Yaskawa INFORM job: R1_W27-A3(90,0)OK-KM.JBI

/JOB
//NAME R1_W27-A3(90,0)OK-KM
///FOLDERNAME KRIS-SCIANA
//POS
///NPOS 43,43,0,3,0,0
///TOOL 0
///POSTYPE PULSE
///PULSE
C00000=4830,83199,5771,6899,94988,75055
C00001=-9773,79383,9827,16212,95277,69552
C00002=-9773,79383,9827,16212,95277,-53372
C00003=-9773,-28468,-43390,16212,95277,-53372
C00004=-118130,28395,29263,-77612,79106,-42908
C00005=-118130,42832,63459,-80282,76069,-36632
C00006=-121022,40509,60957,-80752,74157,-36980
C00007=-122076,40550,60998,-80949,73435,-37043
C00008=-122717,40599,61051,-81070,72994,-37080
C00009=-122076,40550,60998,-80949,73435,-37043
C00010=-122043,47472,68552,-81246,73253,-36526
C00011=-122055,44833,65640,-81126,73325,-36733
C00012=-121022,40509,60957,-80752,74157,-36980
C00013=-118130,28395,29263,-77612,79106,-42908
C00014=-120301,29173,30032,-77655,77552,-43056
C00015=-120039,32113,44650,-90901,76713,-36723
C00016=-120861,32104,44640,-91018,76127,-36728
C00017=-119313,33187,45743,-90820,77231,-36662
C00018=-119853,35892,48525,-90967,76837,-36513
C00019=-119313,33187,45743,-90820,77231,-36662
C00020=-118868,30790,31644,-84323,85642,-41471
C00021=-130429,-11916,41219,-108053,40291,-28638
C00022=-116428,-13316,-7274,-52109,62616,-45524
C00023=-117742,-2204,1538,-51719,62054,-45954
C00024=-115860,2997,30006,-91299,52035,-28528
C00025=-121469,1006,3731,-50735,60158,-46989
C00026=-120227,302,2593,-50891,61069,-46816
C00027=-115745,-1819,28231,-92358,52111,-27726
C00028=-112555,-4087,35757,-96933,59618,-24349
C00029=-112542,-4035,35819,-96942,59654,-24342
C00030=-111238,-10662,2688,-62879,64047,-42529
C00031=-111998,-8144,-211,-53563,64102,-43814
C00032=-114545,-38172,-18809,-58928,38901,31311
C00033=-120615,-32838,-15388,-55575,35611,29062
C00034=-102867,26964,48378,-82054,78500,40282
C00035=-119784,-31977,-14810,-55883,36152,29279
C00036=-120619,-32587,-15219,-55544,35624,29044
C00037=-102846,27333,48386,-82014,78545,40201
C00038=-102203,45516,96371,-91697,68609,49479
C00039=-95028,10215,48172,-86436,71799,45925
C00040=-80780,-67431,-36414,-60607,42164,32637
C00041=-21077,34801,-6145,-35147,72854,61023
C00042=19629,104504,14492,-17788,93778,80377
BC00000=161822,1138,1029509
BC00001=179661,1053,1007237
BC00002=277355,1053,807792
BC00003=277355,1053,807792
BC00004=398174,15,734423
BC00005=398174,15,734423
BC00006=398174,15,734423
BC00007=398174,15,734423
BC00008=398174,15,734423
BC00009=398174,15,734423
BC00010=398174,15,734423
BC00011=398174,15,734423
BC00012=398174,15,734423
BC00013=398174,15,734423
BC00014=398174,15,718477
BC00015=396635,15,712098
BC00016=396635,15,712098
BC00017=396635,15,712098
BC00018=396635,15,712098
BC00019=396635,15,712098
BC00020=398174,10910,727845
BC00021=398174,19843,1075175
BC00022=363223,15,893026
BC00023=359892,15,870362
BC00024=358663,16,873958
BC00025=358560,15,861296
BC00026=358560,15,861296
BC00027=358663,16,873958
BC00028=358610,15,874107
BC00029=358610,15,874108
BC00030=358643,15,874329
BC00031=363273,15,905837
BC00032=348983,15,797430
BC00033=344731,15,795268
BC00034=343031,15,794403
BC00035=343031,15,794403
BC00036=343031,15,794403
BC00037=343031,15,644273
BC00038=343031,15,794403
BC00039=343387,15,790284
BC00040=348817,15,727589
BC00041=229605,324,912929
BC00042=148325,534,1039296
///POSTYPE BASE
///RECTAN
///RCONF 0,0,0,0,1,0,0,0,0,0,0,0,0,0,0,0,0,0,0,0,0,0,0,0
P00006=2.006,1.622,-0.565,0.0000,0.0000,0.0000
///RCONF 0,0,0,0,0,0,0,0,0,0,0,0,0,0,0,0,0,0,0,0,0,0,0,0
P00025=3.643,0.007,-2.585,0.0000,0.0000,0.0000
P00026=2.644,0.055,-2.583,0.0000,0.0000,0.0000
//INST
///DATE 2025/04/11 12:42
///ATTR SC,RW
///GROUP1 RB1,BS1
NOP
SFTOF
MOVJ C00000 BC00000 VJ=100.00
MOVJ C00001 BC00001 VJ=100.00
MOVJ C00002 BC00002 VJ=100.00
MOVJ C00003 BC00003 VJ=100.00
MOVL C00004 BC00004 V=1000.0
MOVL C00005 BC00005 V=1000.0
MOVL C00006 BC00006 V=250.0
MOVL C00007 BC00007 V=100.0
REFP 3 C00008 BC00008
CALL JOB:SEARCH-R1
SET P026 P006
SFTON P026
MOVL C00009 BC00009 V=60.0
REFP 3 C00010 BC00010
CALL JOB:SEARCH-R1
SET P026 P006
SFTON P026
MOVL C00011 BC00011 V=60.0
MOVL C00012 BC00012 V=166.7
SFTOF
MOVL C00013 BC00013 V=1000.0
MOVL C00014 BC00014 V=250.0
MOVL C00015 BC00015 V=100.0
REFP 3 C00016 BC00016
CALL JOB:SEARCH-R1
SET P025 P006
SFTON P025
MOVL C00017 BC00017 V=60.0
REFP 3 C00018 BC00018
CALL JOB:SEARCH-R1
SET P025 P006
SFTON P025
MOVL C00019 BC00019 V=60.0
MOVL C00020 BC00020 V=166.7
'Path VIA1038
SFTOF
MOVL C00021 BC00021 V=333.3
'Path W998
SFTOF
SFTON P025
CALL JOB:COFNIJ_DRUT
MOVJ C00022 BC00022 VJ=100.00
MOVJ C00023 BC00023 VJ=100.00
MOVL C00024 BC00024 V=100.0 PL=0
REFP 1 C00025 BC00025
REFP 2 C00026 BC00026
MACRO1 MJ#(0) ARGF7
ARCON
MOVL C00027 BC00027 V=10.0
COMM MOVL C00028 BC00028 V=11.2
MOVL C00029 BC00029 V=11.2
ARCOF
MOVL C00030 BC00030 V=166.7
MOVL C00031 BC00031 V=166.7
SFTOF
'Path W999
SFTOF
SFTON P025
MOVJ C00032 BC00032 VJ=100.00
MOVJ C00033 BC00033 VJ=100.00
MOVL C00034 BC00034 V=100.0 PL=0
REFP 1 C00035 BC00035
REFP 2 C00036 BC00036
MACRO1 MJ#(0) ARGF7
ARCON
SFTON P026
MOVL C00037 BC00037 V=10.8
ARCOF
MOVL C00038 BC00038 V=250.0
MOVL C00039 BC00039 V=250.0
MOVJ C00040 BC00040 VJ=100.00
SFTOF
MOVJ C00041 BC00041 VJ=100.00
MOVJ C00042 BC00042 VJ=100.00
END
